% RSLogix 500 project CHEMICAL MIXING PROCESS LOGIC.RSS, saved by version 8.30.00.16 %
PROJECT "UNTITLED"    % processor: Bul.1763 MicroLogix 1100 Series B %

PROGRAM FILES
  LAD 2   8 rungs

DATA FILES
  O0 OUTPUT  4 elements
  I1 INPUT  6 elements
  S2 STATUS  66 elements
  B3 BINARY  1 elements
  T4 TIMER  1 elements
  C5 COUNTER  1 elements
  R6 CONTROL  1 elements
  N7 INTEGER  1 elements
  F8 FLOAT  1 elements

LADDER 2
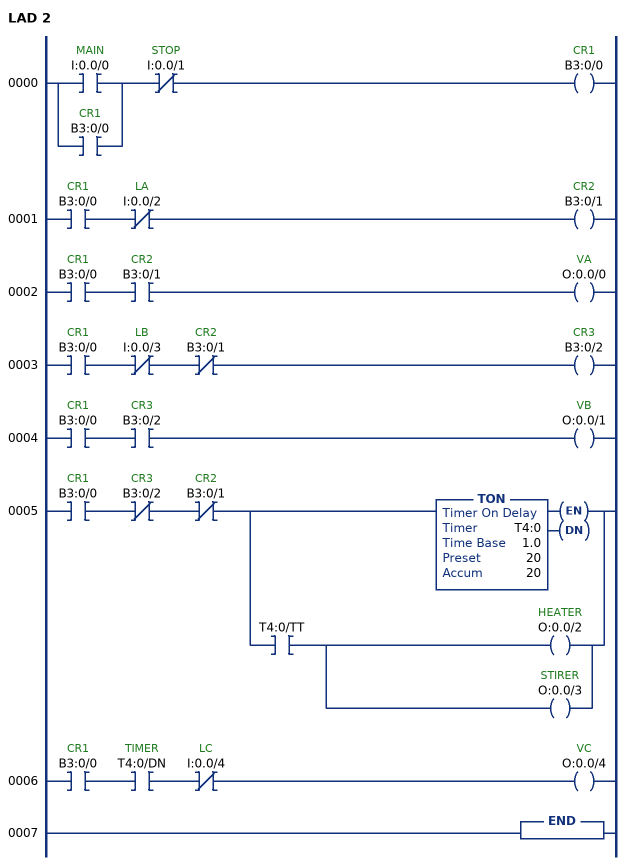
% Rung: 0 %
SOR BST XIC I:0.0/0 NXB XIC B3:0/0 BND XIO I:0.0/1 OTE B3:0/0 EOR
%   I:0.0/0  "MAIN" %
%   B3:0/0  "CR1" %
%   I:0.0/1  "STOP" %
% Rung: 1 %
SOR XIC B3:0/0 XIO I:0.0/2 OTE B3:0/1 EOR
%   B3:0/0  "CR1" %
%   I:0.0/2  "LA" %
%   B3:0/1  "CR2" %
% Rung: 2 %
SOR XIC B3:0/0 XIC B3:0/1 OTE O:0.0/0 EOR
%   B3:0/0  "CR1" %
%   B3:0/1  "CR2" %
%   O:0.0/0  "VA" %
% Rung: 3 %
SOR XIC B3:0/0 XIO I:0.0/3 XIO B3:0/1 OTE B3:0/2 EOR
%   B3:0/0  "CR1" %
%   I:0.0/3  "LB" %
%   B3:0/1  "CR2" %
%   B3:0/2  "CR3" %
% Rung: 4 %
SOR XIC B3:0/0 XIC B3:0/2 OTE O:0.0/1 EOR
%   B3:0/0  "CR1" %
%   B3:0/2  "CR3" %
%   O:0.0/1  "VB" %
% Rung: 5 %
SOR XIC B3:0/0 XIO B3:0/2 XIO B3:0/1 BST TON T4:0 1.0 20 20 NXB XIC T4:0/TT BST OTE O:0.0/2 NXB OTE O:0.0/3 BND BND EOR
%   B3:0/0  "CR1" %
%   B3:0/2  "CR3" %
%   B3:0/1  "CR2" %
%   O:0.0/2  "HEATER" %
%   O:0.0/3  "STIRER" %
% Rung: 6 %
SOR XIC B3:0/0 XIC T4:0/DN XIO I:0.0/4 OTE O:0.0/4 EOR
%   B3:0/0  "CR1" %
%   T4:0/DN  "TIMER" %
%   I:0.0/4  "LC" %
%   O:0.0/4  "VC" %
% Rung: 7 %
SOR END EOR

DATA TABLE (non-zero values as saved)
DATA T4
% .PRE .ACC %
% T4:0 % 20 20
